TYPE csp_transfer_infeed_accU_depth_enum :
(
	CSP_TRANSFER_INFEED_ACCU_DEPTH_STATUS_NOT_INITIALIZED 							:= 0,
	CSP_TRANSFER_INFEED_ACCU_DEPTH_STATUS_DISABLED 									:= 10,
	CSP_TRANSFER_INFEED_ACCU_DEPTH_STATUS_POSITION_CHECK							:= 20,
	CSP_TRANSFER_INFEED_ACCU_DEPTH_STATUS_ENABLE_REQUEST 							:= 30,
	CSP_TRANSFER_INFEED_ACCU_DEPTH_STATUS_ENABLED 									:= 40,
	CSP_TRANSFER_INFEED_ACCU_DEPTH_STATUS_CHECK_MOVE								:= 41,
	CSP_TRANSFER_INFEED_ACCU_DEPTH_STATUS_OUTRUN									:= 42,
	CSP_TRANSFER_INFEED_ACCU_DEPTH_STATUS_WAIT_FOR_OUTRUN							:= 43,
	CSP_TRANSFER_INFEED_ACCU_DEPTH_STATUS_ABS_MOVE_REQUEST							:= 50,
	CSP_TRANSFER_INFEED_ACCU_DEPTH_STATUS_ABS_MOVING								:= 60,
	CSP_TRANSFER_INFEED_ACCU_DEPTH_STATUS_STOP_REQUEST 								:= 70,
	CSP_TRANSFER_INFEED_ACCU_DEPTH_STATUS_DISABLE_REQUEST 							:= 80,
	CSP_TRANSFER_INFEED_ACCU_DEPTH_STATUS_DISABLING 								:= 90
) := CSP_TRANSFER_INFEED_ACCU_DEPTH_STATUS_NOT_INITIALIZED;
END_TYPE

(* stored: Version 1.1.0.1, ProductVersion 3.1.4024.3
   DUT csp_transfer_infeed_accU_depth_enum: Id {f83d726c-9b16-44bc-b515-dffb83109fc3} *)
